{attribute 'qualified_only'}
{attribute 'strict'}
TYPE E_Color :
(
	NoColor := 0,
	Blue,
	Green,
	Yellow
	
);
END_TYPE

(* stored: Version 1.1.0.1, ProductVersion 3.1.4024.12
   DUT E_Color: Id {187cab3c-9d5d-4b15-87e5-3aa7745b6b59} *)
